// Packs color components into ARGB.
FUNCTION GenArgb : Argb
VAR_INPUT
	nRed: USINT; // Red channel.
	nGreen: USINT; // Green channel.
	nBlue: USINT; // Blue channel.
	nAlpha: USINT; // Alpha channel.
END_VAR

GenArgb := USINT_TO_UDINT(nBlue) OR
			SHL(USINT_TO_UDINT(nGreen), 8) OR
			SHL(USINT_TO_UDINT(nRed), 16) OR
			SHL(USINT_TO_UDINT(nAlpha), 24);

END_FUNCTION

(* stored: Version 1.1.0.1
   POU GenArgb: Id {9c58ba81-b5d6-4a9d-8df8-dc2f4420ed2f}, SpecialFunc None *)
